// TIA Portal V18 export
DATA_BLOCK "_BTNS"   // DB3
VERSION : 0.1
// stored: AutoNumber true, DBAccessibleFromOPCUA true, InstanceOfName BTNS_FB, InstanceOfType FB
"BTNS_FB"
   // VAR_INPUT
   //    "remote key activated" : Bool;
   //    xCylceStart : Bool;
   //    xDefectMark : Bool;
   //    xDefectNext : Bool;
   //    xDefectPrev : Bool;
   //    xHome : Bool;
   //    xLaser : Bool;
   //    xLoad : Bool;
   //    xControl1 : Bool;
   //    xControl2 : Bool;
   //    xbDoorsFwdClose : Bool;
   //    xbDoorsRevOpen : Bool;
   //    xbo1Tiltfwd : Bool;
   //    xbo1Tiltrev : Bool;
   //    xbo2RotHome : Bool;
   //    xbo2Rotrev : Bool;
   //    xSwAuto : Bool;
   //    xSwMan : Bool;
   //    xbXfwd : Bool;
   //    xbxrev : Bool;
   //    xbyfwd : Bool;
   //    xbyrev : Bool;
   //    xbzfwd : Bool;
   //    xbzrev : Bool;
   //    xbo2Rotfwd : Bool;
   // END_VAR
   // VAR_OUTPUT
   //    remPowerOut : Bool;
   //    yLedShutter : Bool;
   //    yLedAuto : Bool;
   //    ysirenFinished : Bool;
   //    ySirenError : Bool;
   // END_VAR
   // VAR
   //    desk_yledShutter { S7_SetPoint := 'True'} : "LED_FBD";
   // END_VAR
BEGIN
END_DATA_BLOCK
